{attribute 'qualified_only'}
VAR_GLOBAL


	fbPB1_Wyk1_K1_HMI				: FB_Component_HMI (itfBaseLoggerConnector := GVL.fbLogger, itfComponentConnector := GVL_Variable.fbPB1_Wyk1_K1);
	fbPB1_Wyk1_K2_HMI				: FB_Component_HMI (itfBaseLoggerConnector := GVL.fbLogger, itfComponentConnector := GVL_Variable.fbPB1_Wyk1_K2);
	fbPB1_Wyk1_HMI					: FB_ControlElement_HMI (
										itfBaseLoggerConnector 		:= GVL.fbLogger,
										itfControlElementConnector 	:= GVL_Variable.fbPB1_Wyk1,
										itfComponent1				:= fbPB1_Wyk1_K1_HMI,
										itfComponent2				:= fbPB1_Wyk1_K2_HMI
									);
//	
	fbPB1_Wyk2_K1_HMI				: FB_Component_HMI (itfBaseLoggerConnector := GVL.fbLogger, itfComponentConnector := GVL_Variable.fbPB1_Wyk2_K1);
	fbPB1_Wyk2_K2_HMI				: FB_Component_HMI (itfBaseLoggerConnector := GVL.fbLogger, itfComponentConnector := GVL_Variable.fbPB1_Wyk2_K2);
	fbPB1_Wyk2_HMI					: FB_ControlElement_HMI (
										itfBaseLoggerConnector 		:= GVL.fbLogger,
										itfControlElementConnector 	:= GVL_Variable.fbPB1_Wyk2,
										itfComponent1				:= fbPB1_Wyk2_K1_HMI,
										itfComponent2				:= fbPB1_Wyk2_K2_HMI
									);
//
	fbPB1_ZL1_Wyk1_K1_HMI			: FB_Component_HMI (itfBaseLoggerConnector := GVL.fbLogger, itfComponentConnector := GVL_Variable.fbPB1_ZL1_Wyk1_K1);
	fbPB1_ZL1_Wyk1_K2_HMI			: FB_Component_HMI (itfBaseLoggerConnector := GVL.fbLogger, itfComponentConnector := GVL_Variable.fbPB1_ZL1_Wyk1_K2);
	fbPB1_ZL1_Wyk1_HMI				: FB_ControlElement_HMI (
										itfBaseLoggerConnector 		:= GVL.fbLogger,
										itfControlElementConnector 	:= GVL_Variable.fbPB1_ZL1_Wyk1,
										itfComponent1				:= fbPB1_ZL1_Wyk1_K1_HMI,
										itfComponent2				:= fbPB1_ZL1_Wyk1_K2_HMI
									);
	fbPB1_ZL1_Wyk2_K1_HMI			: FB_Component_HMI (itfBaseLoggerConnector := GVL.fbLogger, itfComponentConnector := GVL_Variable.fbPB1_ZL1_Wyk2_K1);
	fbPB1_ZL1_Wyk2_K2_HMI			: FB_Component_HMI (itfBaseLoggerConnector := GVL.fbLogger, itfComponentConnector := GVL_Variable.fbPB1_ZL1_Wyk2_K2);
	fbPB1_ZL1_Wyk2_HMI				: FB_ControlElement_HMI (
										itfBaseLoggerConnector 		:= GVL.fbLogger,
										itfControlElementConnector 	:= GVL_Variable.fbPB1_ZL1_Wyk2,
										itfComponent1				:= fbPB1_ZL1_Wyk2_K1_HMI,
										itfComponent2				:= fbPB1_ZL1_Wyk2_K2_HMI
									);
	fbPB1_ZL1_K1_HMI				: FB_Component_HMI (itfBaseLoggerConnector := GVL.fbLogger, itfComponentConnector := GVL_Variable.fbPB1_ZL1_K1);
	fbPB1_ZL1_K2_HMI				: FB_Component_HMI (itfBaseLoggerConnector := GVL.fbLogger, itfComponentConnector := GVL_Variable.fbPB1_ZL1_K2);
	fbPB1_ZL1_HMI					: FB_GroupElement_HMI (
										itfBaseLoggerConnector 		:= GVL.fbLogger,
										itfGroupElementConnector 	:= GVL_Variable.fbPB1_ZL1,
										itfControlElement1			:= fbPB1_ZL1_Wyk1_HMI,
										itfControlElement2			:= fbPB1_ZL1_Wyk2_HMI,
										itfComponent1				:= fbPB1_ZL1_K1_HMI,
										itfComponent2				:= fbPB1_ZL1_K2_HMI
									);
	
	fbPB1_K1_HMI					: FB_Component_HMI (itfBaseLoggerConnector := GVL.fbLogger, itfComponentConnector := GVL_Variable.fbPB1_K1);
	fbPB1_K2_HMI					: FB_Component_HMI (itfBaseLoggerConnector := GVL.fbLogger, itfComponentConnector := GVL_Variable.fbPB1_K2);
	fbPB1_K3_HMI					: FB_Component_HMI (itfBaseLoggerConnector := GVL.fbLogger, itfComponentConnector := GVL_Variable.fbPB1_K3);
//	
	fbPB1_HMI						: FB_TopElement_HMI (
										itfBaseLoggerConnector				:= GVL.fbLogger,
                                        itfTopElementConnector				:= GVL_Variable.fbPB1,
                                        itfControlElement1					:= fbPB1_Wyk1_HMI,
                                        itfControlElement2					:= fbPB1_Wyk2_HMI,
                                        itfGroupElement1					:= fbPB1_ZL1_HMI,
                                        itfComponent1						:= fbPB1_K1_HMI,
                                        itfComponent2						:= fbPB1_K2_HMI,
                                        itfComponent3						:= fbPB1_K3_HMI
									);
	
END_VAR

(* stored: Version 1.1.0.1, ProductVersion 3.1.4024.15
   GVL GVL_VariableHMI: Id {b9a94705-a932-4492-af2c-d0486e584051} *)
